(* PLC project  *)

CONFIGURATION Empty_Module_25
END_CONFIGURATION
